SUBAPPLICATION mapping_Uebung_039 (* Spiegelabfolge V2 mit Schrittkette *)
  (* Standard: 61499-2; Description: Copyright (c) 2023 Meisterschulen am Ostbahnhof This program and the accompanying materials are made available under the terms of the Eclipse Public License 2.0 which is available at https://www.eclipse.org/legal/epl-2.0/ SPDX-License-Identifier: EPL-2.0 *)
  (* Version 1.0, 2023-10-23, Franz Höpfinger, Meisterschulen am Ostbahnhof *)
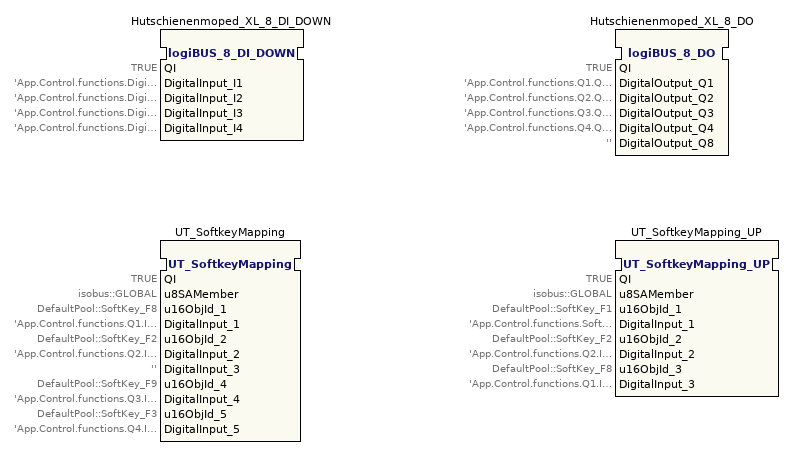
  FBS
    Hutschienenmoped_XL_8_DO : logiBUS_8_DO(QI := TRUE, DigitalOutput_Q1 := 'App.Control.functions.Q1.QX', DigitalOutput_Q2 := 'App.Control.functions.Q2.QX', DigitalOutput_Q3 := 'App.Control.functions.Q3.QX', DigitalOutput_Q4 := 'App.Control.functions.Q4.QX', DigitalOutput_Q8 := '');
    UT_SoftkeyMapping_UP : UT_SoftkeyMapping_UP(QI := TRUE, u8SAMember := isobus::GLOBAL, u16ObjId_1 := DefaultPool::SoftKey_F1, DigitalInput_1 := 'App.Control.functions.SoftKey_F1_UP', u16ObjId_2 := DefaultPool::SoftKey_F2, DigitalInput_2 := 'App.Control.functions.Q2.IE', u16ObjId_3 := DefaultPool::SoftKey_F8, DigitalInput_3 := 'App.Control.functions.Q1.IE');
    Hutschienenmoped_XL_8_DI_DOWN : logiBUS_8_DI_DOWN(QI := TRUE, DigitalInput_I1 := 'App.Control.functions.DigitalInput_DOWN_I1', DigitalInput_I2 := 'App.Control.functions.DigitalInput_DOWN_I2', DigitalInput_I3 := 'App.Control.functions.DigitalInput_DOWN_I3', DigitalInput_I4 := 'App.Control.functions.DigitalInput_DOWN_I4');
    UT_SoftkeyMapping : UT_SoftkeyMapping(QI := TRUE, u8SAMember := isobus::GLOBAL, u16ObjId_1 := DefaultPool::SoftKey_F8, DigitalInput_1 := 'App.Control.functions.Q1.IX', u16ObjId_2 := DefaultPool::SoftKey_F2, DigitalInput_2 := 'App.Control.functions.Q2.IX', DigitalInput_3 := '', u16ObjId_4 := DefaultPool::SoftKey_F9, DigitalInput_4 := 'App.Control.functions.Q3.IX', u16ObjId_5 := DefaultPool::SoftKey_F3, DigitalInput_5 := 'App.Control.functions.Q4.IX');
  END_FBS
END_SUBAPPLICATION
